(* IEC 61131-3 sources: programs/VI-54/VI-54_20171205/VI-54_20171205/Stations/Screen/LseClass170718/Class/SyncTimeHMI, 1 file *)

(* ---- SyncTimeHMI.st ---- *)
(*!
<Class
	Name               = "SyncTimeHMI"
	Revision           = "1.0"
	RealtimeTask       = "false"
	CyclicTask         = "false"
	BackgroundTask     = "false"
	Sigmatek           = "false"
	OSInterface        = "false"
	HighPriority       = "false"
	Automatic          = "false"
	UpdateMode         = "Prescan"
	SharedCommandTable = "true"
	Objectsize         = "(540,180)"
	Comment            = "class reads date and time from two clients (within the adjusted zycletime)&#13;&#10;and writes these values to the servers">
	<Channels>
		<Server Name="sSyncDate" Visualized="true" Remotely="true" Initialize="false" WriteProtected="true" Retentive="false" Comment="server for sync date"/>
		<Server Name="sSyncTime" Visualized="true" Remotely="true" Initialize="false" WriteProtected="true" Retentive="false" Comment="server for sync time"/>
		<Client Name="ActDate" Required="true" Internal="false" Comment="actual date"/>
		<Client Name="ActTime" Required="true" Internal="false" Comment="actual time"/>
	</Channels>
	<RevDoku>
		<Owner Company="Sigmatek"/>
		<Dokumentation Revision="1.0" Date="2015-11-11" Author="hötant" Company="Sigmatek" Description="creation of class"/>
	</RevDoku>
</Class>
*)
SyncTimeHMI : CLASS
  //Servers:
	sSyncDate 	: SvrChCmd_HDINT;
	sSyncTime 	: SvrCh_HDINT;
  //Clients:
	ActDate 	: CltCh_HDINT;
	ActTime 	: CltCh_HDINT;
  //Variables:
  //Functions:

	FUNCTION VIRTUAL GLOBAL sSyncDate::Read
		VAR_OUTPUT
			output (EAX) 	: HDINT;
		END_VAR;

	FUNCTION VIRTUAL GLOBAL sSyncTime::Read
		VAR_OUTPUT
			output (EAX) 	: HDINT;
		END_VAR;
  //Tables:
	FUNCTION @STD
		VAR_OUTPUT
			ret_code	: CONFSTATES;
		END_VAR;
	FUNCTION GLOBAL TAB @CT_;
END_CLASS;

FUNCTION VIRTUAL GLOBAL SyncTimeHMI::sSyncDate::Read
	VAR_OUTPUT
		output (EAX) 	: HDINT;
	END_VAR

	output := sSyncDate := ActDate := ActDate.Read();

END_FUNCTION

FUNCTION VIRTUAL GLOBAL SyncTimeHMI::sSyncTime::Read
	VAR_OUTPUT
		output (EAX) 	: HDINT;
	END_VAR

	output := sSyncTime :=ActTime :=  ActTime.Read();

END_FUNCTION
